SUBAPPLICATION Uebung_093 (* Beispiel für E_TABLE *)
  (* Standard: 61499-2; Description: Copyright (c) 2023 Meisterschulen am Ostbahnhof This program and the accompanying materials are made available under the terms of the Eclipse Public License 2.0 which is available at https://www.eclipse.org/legal/epl-2.0/ SPDX-License-Identifier: EPL-2.0 *)
  (* Version 1.0, 2023-10-23, Franz Höpfinger, Meisterschulen am Ostbahnhof *)
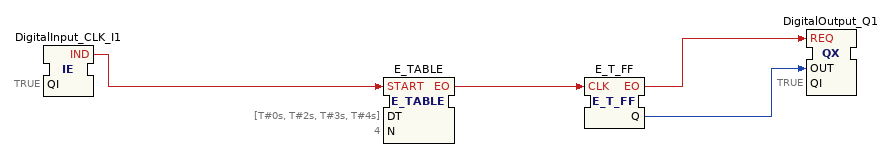
  (* E_TABLE wird 4 Events ausgeben, das erste sofort nach dem Click, das letzte 9s nach dem Click [T#0s, T#2s, T#3s, T#4s] *)
  FBS
    DigitalOutput_Q1 : QX(QI := TRUE);
    E_TABLE : E_TABLE(DT := [T#0s, T#2s, T#3s, T#4s], N := 4);
    DigitalInput_CLK_I1 : IE(QI := TRUE);
    E_T_FF : E_T_FF;
  END_FBS
  EVENT_CONNECTIONS
    DigitalInput_CLK_I1.IND TO E_TABLE.START;
    E_TABLE.EO TO E_T_FF.CLK;
    E_T_FF.EO TO DigitalOutput_Q1.REQ;
  END_CONNECTIONS
  DATA_CONNECTIONS
    E_T_FF.Q TO DigitalOutput_Q1.OUT;
  END_CONNECTIONS
END_SUBAPPLICATION
